(* IEC 61131-3 sources: com.logicals.lc3.webinar/usRTS_RPMControl_iSOC/src_FB_LIB_SAFE/Select, 15 files *)

(* ---- wSEL_BOOL.iecst ---- *)
NAMESPACE logicals.web.standard
NAMESPACE select

/*
 * Function block wrapper for IEC 61131-3 SEL<br>
 * G = selector (BOOL)<br>
 * IN0 = first value (BOOL)<br>
 * IN1 = second value (BOOL)<br>
 * OUT := G ? IN1 : IN0; (BOOL)<br>
 */
FUNCTION_BLOCK wSEL_BOOL
	{ vNameAlignment:="center"; altName:="SEL"; bgColor:="MediumBlue"; width:=120; }
	VAR_INPUT
		G : BOOL;
		IN0 : BOOL;
		IN1 : BOOL;
	END_VAR
	VAR_OUTPUT
		OUT : BOOL;
	END_VAR

	OUT := SEL_BOOL(G:=G, IN0:=IN0, IN1:=IN1, ENO=>ENO);
END_FUNCTION_BLOCK

END_NAMESPACE
END_NAMESPACE

(* ---- wSEL_BYTE.iecst ---- *)
NAMESPACE logicals.web.standard
NAMESPACE select

/*
 * Function block wrapper for IEC 61131-3 SEL<br>
 * G = selector (BOOL)<br>
 * IN0 = first value (BYTE)<br>
 * IN1 = second value (BYTE)<br>
 * OUT := G ? IN1 : IN0; (BYTE)<br>
 */
FUNCTION_BLOCK wSEL_BYTE
	{ vNameAlignment:="center"; altName:="SEL"; bgColor:="DodgerBlue"; width:=120; }
	VAR_INPUT
		G : BOOL;
		IN0 : BYTE;
		IN1 : BYTE;
	END_VAR
	VAR_OUTPUT
		OUT : BYTE;
	END_VAR

	OUT := SEL_BYTE(G:=G, IN0:=IN0, IN1:=IN1, ENO=>ENO);
END_FUNCTION_BLOCK

END_NAMESPACE
END_NAMESPACE

(* ---- wSEL_DINT.iecst ---- *)
NAMESPACE logicals.web.standard
NAMESPACE select

/*
 * Function block wrapper for IEC 61131-3 SEL<br>
 * G = selector (BOOL)<br>
 * IN0 = first value (DINT)<br>
 * IN1 = second value (DINT)<br>
 * OUT := G ? IN1 : IN0; (DINT)<br>
 */
FUNCTION_BLOCK wSEL_DINT
	{ vNameAlignment:="center"; altName:="SEL"; bgColor:="LightPink"; width:=120; }
	VAR_INPUT
		G : BOOL;
		IN0 : DINT;
		IN1 : DINT;
	END_VAR
	VAR_OUTPUT
		OUT : DINT;
	END_VAR

	OUT := SEL_DINT(G:=G, IN0:=IN0, IN1:=IN1, ENO=>ENO);
END_FUNCTION_BLOCK

END_NAMESPACE
END_NAMESPACE

(* ---- wSEL_DWORD.iecst ---- *)
NAMESPACE logicals.web.standard
NAMESPACE select

/*
 * Function block wrapper for IEC 61131-3 SEL<br>
 * G = selector (BOOL)<br>
 * IN0 = first value (DWORD)<br>
 * IN1 = second value (DWORD)<br>
 * OUT := G ? IN1 : IN0; (DWORD)<br>
 */
FUNCTION_BLOCK wSEL_DWORD
	{ vNameAlignment:="center"; altName:="SEL"; bgColor:="DodgerBlue"; width:=120; }
	VAR_INPUT
		G : BOOL;
		IN0 : DWORD;
		IN1 : DWORD;
	END_VAR
	VAR_OUTPUT
		OUT : DWORD;
	END_VAR

	OUT := SEL_DWORD(G:=G, IN0:=IN0, IN1:=IN1, ENO=>ENO);
END_FUNCTION_BLOCK

END_NAMESPACE
END_NAMESPACE

(* ---- wSEL_INT.iecst ---- *)
NAMESPACE logicals.web.standard
NAMESPACE select

/*
 * Function block wrapper for IEC 61131-3 SEL<br>
 * G = selector (BOOL)<br>
 * IN0 = first value (INT)<br>
 * IN1 = second value (INT)<br>
 * OUT := G ? IN1 : IN0; (INT)<br>
 */
FUNCTION_BLOCK wSEL_INT
	{ vNameAlignment:="center"; altName:="SEL"; bgColor:="LightPink"; width:=120; }
	VAR_INPUT
		G : BOOL;
		IN0 : INT;
		IN1 : INT;
	END_VAR
	VAR_OUTPUT
		OUT : INT;
	END_VAR

	OUT := SEL_INT(G:=G, IN0:=IN0, IN1:=IN1, ENO=>ENO);
END_FUNCTION_BLOCK

END_NAMESPACE
END_NAMESPACE

(* ---- wSEL_LINT.iecst ---- *)
NAMESPACE logicals.web.standard
NAMESPACE select

/*
 * Function block wrapper for IEC 61131-3 SEL<br>
 * G = selector (BOOL)<br>
 * IN0 = first value (LINT)<br>
 * IN1 = second value (LINT)<br>
 * OUT := G ? IN1 : IN0; (LINT)<br>
 */
FUNCTION_BLOCK wSEL_LINT
	{ vNameAlignment:="center"; altName:="SEL"; bgColor:="LightPink"; width:=120; }
	VAR_INPUT
		G : BOOL;
		IN0 : LINT;
		IN1 : LINT;
	END_VAR
	VAR_OUTPUT
		OUT : LINT;
	END_VAR

	OUT := SEL_LINT(G:=G, IN0:=IN0, IN1:=IN1, ENO=>ENO);
END_FUNCTION_BLOCK

END_NAMESPACE
END_NAMESPACE

(* ---- wSEL_LREAL.iecst ---- *)
NAMESPACE logicals.web.standard
NAMESPACE select

/*
 * Function block wrapper for IEC 61131-3 SEL<br>
 * G = selector (BOOL)<br>
 * IN0 = first value (LREAL)<br>
 * IN1 = second value (LREAL)<br>
 * OUT := G ? IN1 : IN0; (LREAL)<br>
 */
FUNCTION_BLOCK wSEL_LREAL
	{ vNameAlignment:="center"; altName:="SEL"; bgColor:="Orange"; width:=120; }
	VAR_INPUT
		G : BOOL;
		IN0 : LREAL;
		IN1 : LREAL;
	END_VAR
	VAR_OUTPUT
		OUT : LREAL;
	END_VAR

	OUT := SEL_LREAL(G:=G, IN0:=IN0, IN1:=IN1, ENO=>ENO);
END_FUNCTION_BLOCK

END_NAMESPACE
END_NAMESPACE

(* ---- wSEL_LWORD.iecst ---- *)
NAMESPACE logicals.web.standard
NAMESPACE select

/*
 * Function block wrapper for IEC 61131-3 SEL<br>
 * G = selector (BOOL)<br>
 * IN0 = first value (LWORD)<br>
 * IN1 = second value (LWORD)<br>
 * OUT := G ? IN1 : IN0; (LWORD)<br>
 */
FUNCTION_BLOCK wSEL_LWORD
	{ vNameAlignment:="center"; altName:="SEL"; bgColor:="DodgerBlue"; width:=120; }
	VAR_INPUT
		G : BOOL;
		IN0 : LWORD;
		IN1 : LWORD;
	END_VAR
	VAR_OUTPUT
		OUT : LWORD;
	END_VAR

	OUT := SEL_LWORD(G:=G, IN0:=IN0, IN1:=IN1, ENO=>ENO);
END_FUNCTION_BLOCK

END_NAMESPACE
END_NAMESPACE

(* ---- wSEL_REAL.iecst ---- *)
NAMESPACE logicals.web.standard
NAMESPACE select

/*
 * Function block wrapper for IEC 61131-3 SEL<br>
 * G = selector (BOOL)<br>
 * IN0 = first value (REAL)<br>
 * IN1 = second value (REAL)<br>
 * OUT := G ? IN1 : IN0; (REAL)<br>
 */
FUNCTION_BLOCK wSEL_REAL
	{ vNameAlignment:="center"; altName:="SEL"; bgColor:="Orange"; width:=120; }
	VAR_INPUT
		G : BOOL;
		IN0 : REAL;
		IN1 : REAL;
	END_VAR
	VAR_OUTPUT
		OUT : REAL;
	END_VAR

	OUT := SEL_REAL(G:=G, IN0:=IN0, IN1:=IN1, ENO=>ENO);
END_FUNCTION_BLOCK

END_NAMESPACE
END_NAMESPACE

(* ---- wSEL_SINT.iecst ---- *)
NAMESPACE logicals.web.standard
NAMESPACE select

/*
 * Function block wrapper for IEC 61131-3 SEL<br>
 * G = selector (BOOL)<br>
 * IN0 = first value (SINT)<br>
 * IN1 = second value (SINT)<br>
 * OUT := G ? IN1 : IN0; (SINT)<br>
 */
FUNCTION_BLOCK wSEL_SINT
	{ vNameAlignment:="center"; altName:="SEL"; bgColor:="LightPink"; width:=120; }
	VAR_INPUT
		G : BOOL;
		IN0 : SINT;
		IN1 : SINT;
	END_VAR
	VAR_OUTPUT
		OUT : SINT;
	END_VAR

	OUT := SEL_SINT(G:=G, IN0:=IN0, IN1:=IN1, ENO=>ENO);
END_FUNCTION_BLOCK

END_NAMESPACE
END_NAMESPACE

(* ---- wSEL_UDINT.iecst ---- *)
NAMESPACE logicals.web.standard
NAMESPACE select

/*
 * Function block wrapper for IEC 61131-3 SEL<br>
 * G = selector (BOOL)<br>
 * IN0 = first value (UDINT)<br>
 * IN1 = second value (UDINT)<br>
 * OUT := G ? IN1 : IN0; (UDINT)<br>
 */
FUNCTION_BLOCK wSEL_UDINT
	{ vNameAlignment:="center"; altName:="SEL"; bgColor:="Plum"; width:=120; }
	VAR_INPUT
		G : BOOL;
		IN0 : UDINT;
		IN1 : UDINT;
	END_VAR
	VAR_OUTPUT
		OUT : UDINT;
	END_VAR

	OUT := SEL_UDINT(G:=G, IN0:=IN0, IN1:=IN1, ENO=>ENO);
END_FUNCTION_BLOCK

END_NAMESPACE
END_NAMESPACE

(* ---- wSEL_UINT.iecst ---- *)
NAMESPACE logicals.web.standard
NAMESPACE select

/*
 * Function block wrapper for IEC 61131-3 SEL<br>
 * G = selector (BOOL)<br>
 * IN0 = first value (UINT)<br>
 * IN1 = second value (UINT)<br>
 * OUT := G ? IN1 : IN0; (UINT)<br>
 */
FUNCTION_BLOCK wSEL_UINT
	{ vNameAlignment:="center"; altName:="SEL"; bgColor:="Plum"; width:=120; }
	VAR_INPUT
		G : BOOL;
		IN0 : UINT;
		IN1 : UINT;
	END_VAR
	VAR_OUTPUT
		OUT : UINT;
	END_VAR

	OUT := SEL_UINT(G:=G, IN0:=IN0, IN1:=IN1, ENO=>ENO);
END_FUNCTION_BLOCK

END_NAMESPACE
END_NAMESPACE

(* ---- wSEL_ULINT.iecst ---- *)
NAMESPACE logicals.web.standard
NAMESPACE select

/*
 * Function block wrapper for IEC 61131-3 SEL<br>
 * G = selector (BOOL)<br>
 * IN0 = first value (ULINT)<br>
 * IN1 = second value (ULINT)<br>
 * OUT := G ? IN1 : IN0; (ULINT)<br>
 */
FUNCTION_BLOCK wSEL_ULINT
	{ vNameAlignment:="center"; altName:="SEL"; bgColor:="Plum"; width:=120; }
	VAR_INPUT
		G : BOOL;
		IN0 : ULINT;
		IN1 : ULINT;
	END_VAR
	VAR_OUTPUT
		OUT : ULINT;
	END_VAR

	OUT := SEL_ULINT(G:=G, IN0:=IN0, IN1:=IN1, ENO=>ENO);
END_FUNCTION_BLOCK

END_NAMESPACE
END_NAMESPACE

(* ---- wSEL_USINT.iecst ---- *)
NAMESPACE logicals.web.standard
NAMESPACE select

/*
 * Function block wrapper for IEC 61131-3 SEL<br>
 * G = selector (BOOL)<br>
 * IN0 = first value (USINT)<br>
 * IN1 = second value (USINT)<br>
 * OUT := G ? IN1 : IN0; (USINT)<br>
 */
FUNCTION_BLOCK wSEL_USINT
	{ vNameAlignment:="center"; altName:="SEL"; bgColor:="Plum"; width:=120; }
	VAR_INPUT
		G : BOOL;
		IN0 : USINT;
		IN1 : USINT;
	END_VAR
	VAR_OUTPUT
		OUT : USINT;
	END_VAR

	OUT := SEL_USINT(G:=G, IN0:=IN0, IN1:=IN1, ENO=>ENO);
END_FUNCTION_BLOCK

END_NAMESPACE
END_NAMESPACE

(* ---- wSEL_WORD.iecst ---- *)
NAMESPACE logicals.web.standard
NAMESPACE select

/*
 * Function block wrapper for IEC 61131-3 SEL<br>
 * G = selector (BOOL)<br>
 * IN0 = first value (WORD)<br>
 * IN1 = second value (WORD)<br>
 * OUT := G ? IN1 : IN0; (WORD)<br>
 */
FUNCTION_BLOCK wSEL_WORD
	{ vNameAlignment:="center"; altName:="SEL"; bgColor:="DodgerBlue"; width:=120; }
	VAR_INPUT
		G : BOOL;
		IN0 : WORD;
		IN1 : WORD;
	END_VAR
	VAR_OUTPUT
		OUT : WORD;
	END_VAR

	OUT := SEL_WORD(G:=G, IN0:=IN0, IN1:=IN1, ENO=>ENO);
END_FUNCTION_BLOCK

END_NAMESPACE
END_NAMESPACE
